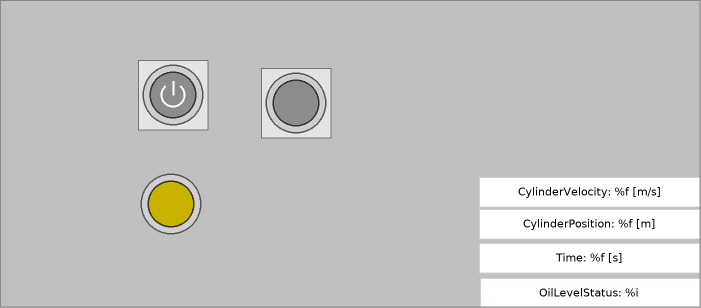
VISUALIZATION Visualization  // 701x308
    PowerSwitch (138,60 70x70), variable: Inputs.bStart, behaviour: TOGGLE, style: Switch-PowerSwitch-Gray
    Lamp1 (136,169 70x70), variable: Outputs.bSimRunning, style: Lamp-Lamp1-Yellow
    Textfield (479,177 221x30), "CylinderVelocity: %f [m/s]", text variable: Outputs.fCylinderVelocity
    Textfield (479,209 221x30), "CylinderPosition: %f [m]", text variable: Outputs.fCylinderPosition
    PushSwitch (261,68 70x70), variable: Inputs.bReset, behaviour: TOGGLE, style: Switch-PushSwitch-Gray
    Textfield (479,243 221x30), "Time: %f [s]", text variable: CraneSimulation.fTime
    Textfield (480,278 221x30), "OilLevelStatus: %i", text variable: CraneSimulation.eOilLevelAlarms
END_VISUALIZATION

(* stored: Version 1.1.0.1, ProductVersion 3.1.4024.10
   Visu Visualization: Id {d64cf4ef-9c3e-41ec-8a01-92d86b637f66} *)
